FUNCTION WRITE_PROTECTED_WORD
VAR_INPUT
    Ptr : POINTER TO WORD;
    Value : WORD;
END_VAR

Ptr^ := Value;

END_FUNCTION

(* stored: Version 1.1.0.1, ProductVersion 3.1.4024.9
   POU WRITE_PROTECTED_WORD: Id {7958aecd-9f81-09a2-1a35-bb6dd127121b}, SpecialFunc None *)
